TYPE U_TRANSLATE_OUT :
UNION
	nArray :	ARRAY[0..15] OF BYTE;
	Label :		S_NAMES_OUT;
END_UNION
END_TYPE

(* stored: Version 1.1.0.1, ProductVersion 3.1.4024.6
   DUT U_TRANSLATE_OUT: Id {7b02a186-d044-474f-9680-9daa8c84f412} *)
